PROGRAM Input_Buffering_RB
VAR PERSISTENT
	
	StackerPartPresentTon: TON;
	StackerPinExtendedTon: TON;
	StackerPinRetractedTon: TON;
	IndexerPartPresentTon: TON;
    SawExtendedTon: TON;
	SawRetractedTon: TON;
	SawClampExtendedTon: TON;
	SawClampRetractedTon: TON;
	SawClampOpenTon: TON;
	SawClampClosedTon: TON;
	TransferClampOpenTon: TON;
	TransferClampClosedTon: TON;
	TransferClampExtdTon: TON;
	TransferClampRetdTon: TON;
	TransferExtdTon: TON;
	TransferRetdTon: TON;
	RibHoistUpTon: TON;
	RibHoistDownTon: TON;
	EjectExtendedTon: TON;
	EjectRetractedTon: TON;
	AirPressureSwitchTon: TON;
	IndexerHomeTon: TON;
	
END_VAR

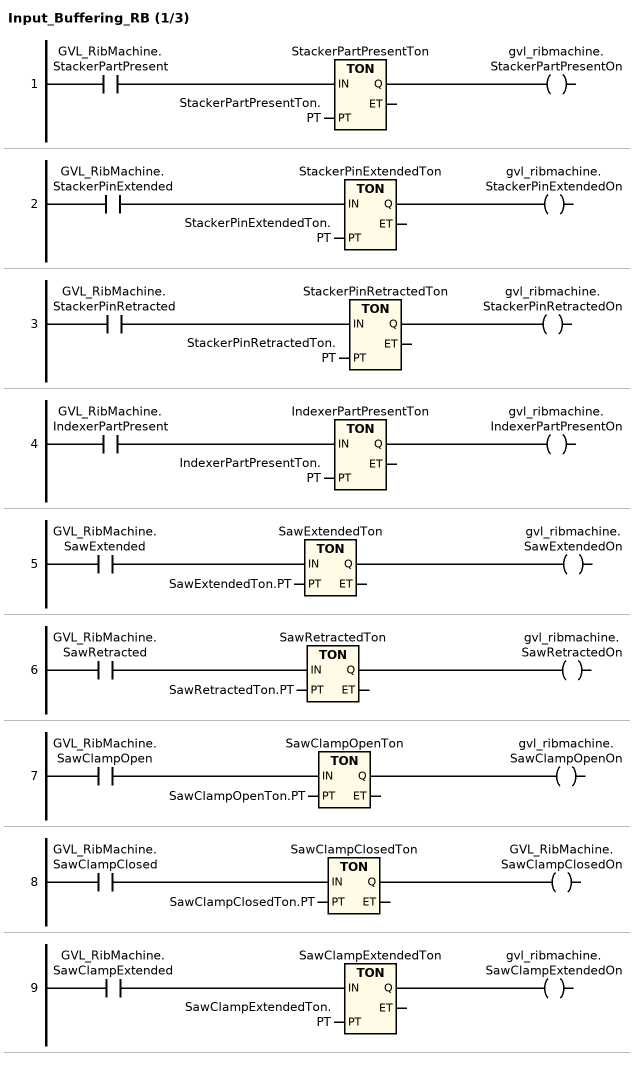
// NETWORK 1
StackerPartPresentTon(IN := GVL_RibMachine.StackerPartPresent, PT := StackerPartPresentTon.PT); // TON
gvl_ribmachine.StackerPartPresentOn := StackerPartPresentTon.Q;

// NETWORK 2
StackerPinExtendedTon(IN := GVL_RibMachine.StackerPinExtended, PT := StackerPinExtendedTon.PT); // TON
gvl_ribmachine.StackerPinExtendedOn := StackerPinExtendedTon.Q;

// NETWORK 3
StackerPinRetractedTon(IN := GVL_RibMachine.StackerPinRetracted, PT := StackerPinRetractedTon.PT); // TON
gvl_ribmachine.StackerPinRetractedOn := StackerPinRetractedTon.Q;

// NETWORK 4
IndexerPartPresentTon(IN := GVL_RibMachine.IndexerPartPresent, PT := IndexerPartPresentTon.PT); // TON
gvl_ribmachine.IndexerPartPresentOn := IndexerPartPresentTon.Q;

// NETWORK 5
SawExtendedTon(IN := GVL_RibMachine.SawExtended, PT := SawExtendedTon.PT); // TON
gvl_ribmachine.SawExtendedOn := SawExtendedTon.Q;

// NETWORK 6
SawRetractedTon(IN := GVL_RibMachine.SawRetracted, PT := SawRetractedTon.PT); // TON
gvl_ribmachine.SawRetractedOn := SawRetractedTon.Q;

// NETWORK 7
SawClampOpenTon(IN := GVL_RibMachine.SawClampOpen, PT := SawClampOpenTon.PT); // TON
gvl_ribmachine.SawClampOpenOn := SawClampOpenTon.Q;

// NETWORK 8
SawClampClosedTon(IN := GVL_RibMachine.SawClampClosed, PT := SawClampClosedTon.PT); // TON
GVL_RibMachine.SawClampClosedOn := SawClampClosedTon.Q;

// NETWORK 9
SawClampExtendedTon(IN := GVL_RibMachine.SawClampExtended, PT := SawClampExtendedTon.PT); // TON
gvl_ribmachine.SawClampExtendedOn := SawClampExtendedTon.Q;

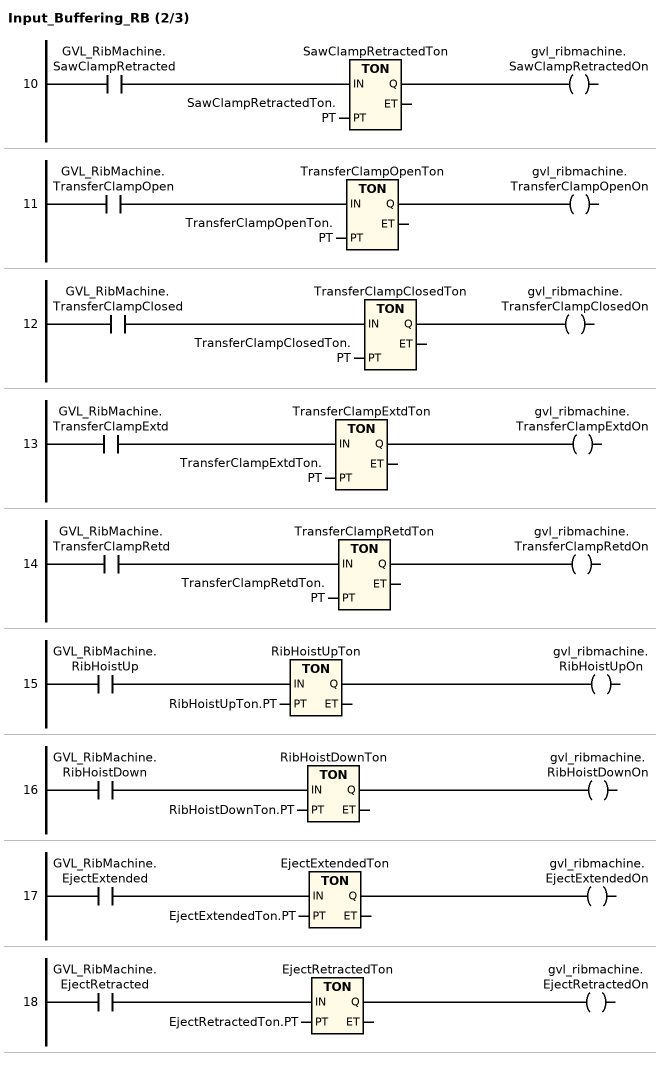
// NETWORK 10
SawClampRetractedTon(IN := GVL_RibMachine.SawClampRetracted, PT := SawClampRetractedTon.PT); // TON
gvl_ribmachine.SawClampRetractedOn := SawClampRetractedTon.Q;

// NETWORK 11
TransferClampOpenTon(IN := GVL_RibMachine.TransferClampOpen, PT := TransferClampOpenTon.PT); // TON
gvl_ribmachine.TransferClampOpenOn := TransferClampOpenTon.Q;

// NETWORK 12
TransferClampClosedTon(IN := GVL_RibMachine.TransferClampClosed, PT := TransferClampClosedTon.PT); // TON
gvl_ribmachine.TransferClampClosedOn := TransferClampClosedTon.Q;

// NETWORK 13
TransferClampExtdTon(IN := GVL_RibMachine.TransferClampExtd, PT := TransferClampExtdTon.PT); // TON
gvl_ribmachine.TransferClampExtdOn := TransferClampExtdTon.Q;

// NETWORK 14
TransferClampRetdTon(IN := GVL_RibMachine.TransferClampRetd, PT := TransferClampRetdTon.PT); // TON
gvl_ribmachine.TransferClampRetdOn := TransferClampRetdTon.Q;

// NETWORK 15
RibHoistUpTon(IN := GVL_RibMachine.RibHoistUp, PT := RibHoistUpTon.PT); // TON
gvl_ribmachine.RibHoistUpOn := RibHoistUpTon.Q;

// NETWORK 16
RibHoistDownTon(IN := GVL_RibMachine.RibHoistDown, PT := RibHoistDownTon.PT); // TON
gvl_ribmachine.RibHoistDownOn := RibHoistDownTon.Q;

// NETWORK 17
EjectExtendedTon(IN := GVL_RibMachine.EjectExtended, PT := EjectExtendedTon.PT); // TON
gvl_ribmachine.EjectExtendedOn := EjectExtendedTon.Q;

// NETWORK 18
EjectRetractedTon(IN := GVL_RibMachine.EjectRetracted, PT := EjectRetractedTon.PT); // TON
gvl_ribmachine.EjectRetractedOn := EjectRetractedTon.Q;

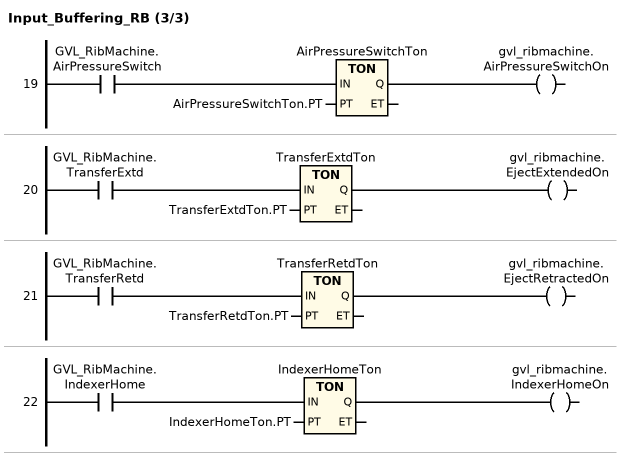
// NETWORK 19
AirPressureSwitchTon(IN := GVL_RibMachine.AirPressureSwitch, PT := AirPressureSwitchTon.PT); // TON
gvl_ribmachine.AirPressureSwitchOn := AirPressureSwitchTon.Q;

// NETWORK 20
TransferExtdTon(IN := GVL_RibMachine.TransferExtd, PT := TransferExtdTon.PT); // TON
gvl_ribmachine.EjectExtendedOn := TransferExtdTon.Q;

// NETWORK 21
TransferRetdTon(IN := GVL_RibMachine.TransferRetd, PT := TransferRetdTon.PT); // TON
gvl_ribmachine.EjectRetractedOn := TransferRetdTon.Q;

// NETWORK 22
IndexerHomeTon(IN := GVL_RibMachine.IndexerHome, PT := IndexerHomeTon.PT); // TON
gvl_ribmachine.IndexerHomeOn := IndexerHomeTon.Q;

END_PROGRAM

(* stored: Version 1.1.0.1, ProductVersion 3.1.4024.12
   POU Input_Buffering_RB: Id {c10cecad-b7c1-4bfc-8dfe-b90a21ed54f4}, SpecialFunc None *)
